FUNCTION_BLOCK FB_Auto_SC
VAR_INPUT
	bEnable				: BOOL;
END_VAR
VAR_OUTPUT
	fPCV				: LREAL;
	fSCV				: LREAL;
	
END_VAR
VAR
	
//Function Blocks
fbPID_payloadpos			: FB_PID_Controller_posref;
fbDeadband_startpos			: FB_Deadband_Auto;
fbDeadband					: FB_Deadband;
fbDisplacementControl_SC	: FB_DisplacementControl_SC;
fbDerivator					: FB_Derivator;

fbClock						: FB_Clock;
fbMUX_selector				: FB_MUX_selector;

//Deadband
fUpperdeadband				: LREAL := 0.5;
fLowerdeadband				: LREAL := 0.14;
fNeutraldeadband			: LREAL := 0.35;
fDeadbandComp_out			: LREAL;

//Outer Loop output
fSC_ClosedLoopSingal		: LREAL;

//VelRef
fWinchVelRefSine			: LREAL;

//Valvesignals
fPCV_set					: LREAL := 1.0;
fPCV_On						: LREAL;
fPCV_Off					: LREAL;

fSCV_startpos				: LREAL;
fSCV_sine					: LREAL;
fSCV_Off					: LREAL;


END_VAR
VAR // added by the converter: edge detectors and wires of the graphical bodies
    _w1 : LREAL;
    _w2 : BOOL;
END_VAR

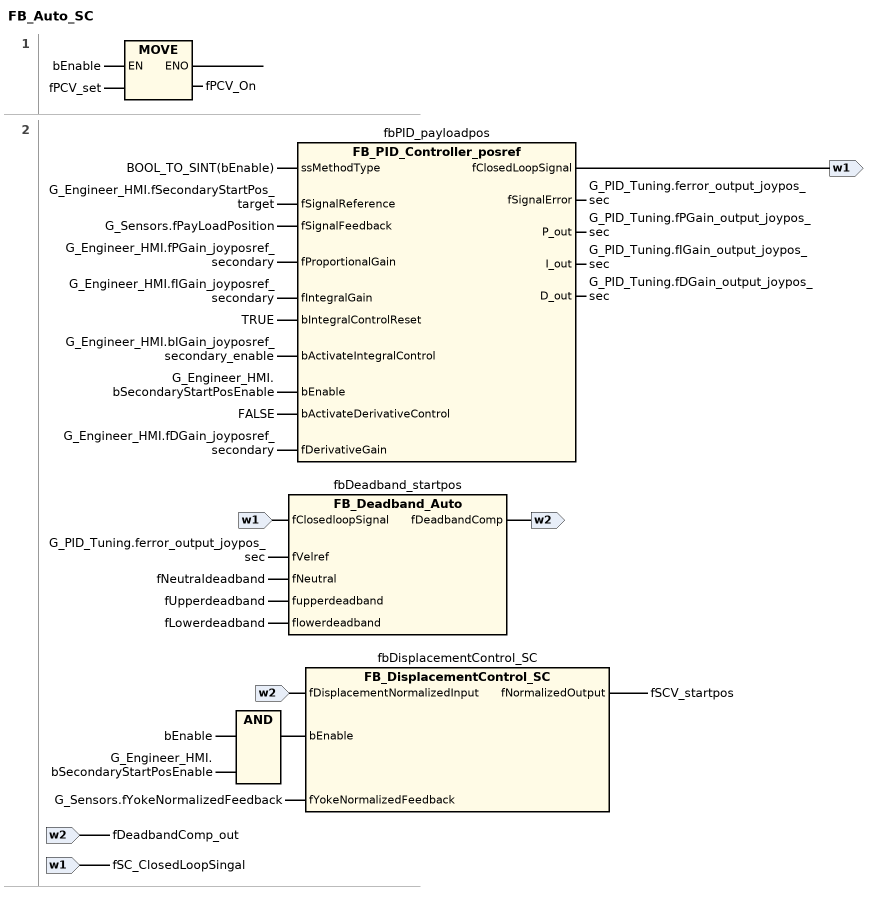
// NETWORK 1
IF bEnable THEN fPCV_On := fPCV_set; END_IF

// NETWORK 2
fbPID_payloadpos(
    ssMethodType := BOOL_TO_SINT(bEnable),
    fSignalReference := G_Engineer_HMI.fSecondaryStartPos_target,
    fSignalFeedback := G_Sensors.fPayLoadPosition,
    fProportionalGain := G_Engineer_HMI.fPGain_joyposref_secondary,
    fIntegralGain := G_Engineer_HMI.fIGain_joyposref_secondary,
    bIntegralControlReset := TRUE,
    bActivateIntegralControl := G_Engineer_HMI.bIGain_joyposref_secondary_enable,
    bEnable := G_Engineer_HMI.bSecondaryStartPosEnable,
    bActivateDerivativeControl := FALSE,
    fDerivativeGain := G_Engineer_HMI.fDGain_joyposref_secondary,
    fSignalError => G_PID_Tuning.ferror_output_joypos_sec,
    P_out => G_PID_Tuning.fPGain_output_joypos_sec,
    I_out => G_PID_Tuning.fIGain_output_joypos_sec,
    D_out => G_PID_Tuning.fDGain_output_joypos_sec); // FB_PID_Controller_posref
fbDeadband_startpos(
    fClosedloopSignal := fbPID_payloadpos.fClosedLoopSignal,
    fVelref := G_PID_Tuning.ferror_output_joypos_sec,
    fNeutral := fNeutraldeadband,
    fupperdeadband := fUpperdeadband,
    flowerdeadband := fLowerdeadband); // FB_Deadband_Auto
fbDisplacementControl_SC(
    fDisplacementNormalizedInput := fbDeadband_startpos.fDeadbandComp,
    bEnable := bEnable AND G_Engineer_HMI.bSecondaryStartPosEnable,
    fYokeNormalizedFeedback := G_Sensors.fYokeNormalizedFeedback); // FB_DisplacementControl_SC
fSCV_startpos := fbDisplacementControl_SC.fNormalizedOutput;
fDeadbandComp_out := fbDeadband_startpos.fDeadbandComp;
fSC_ClosedLoopSingal := fbPID_payloadpos.fClosedLoopSignal;

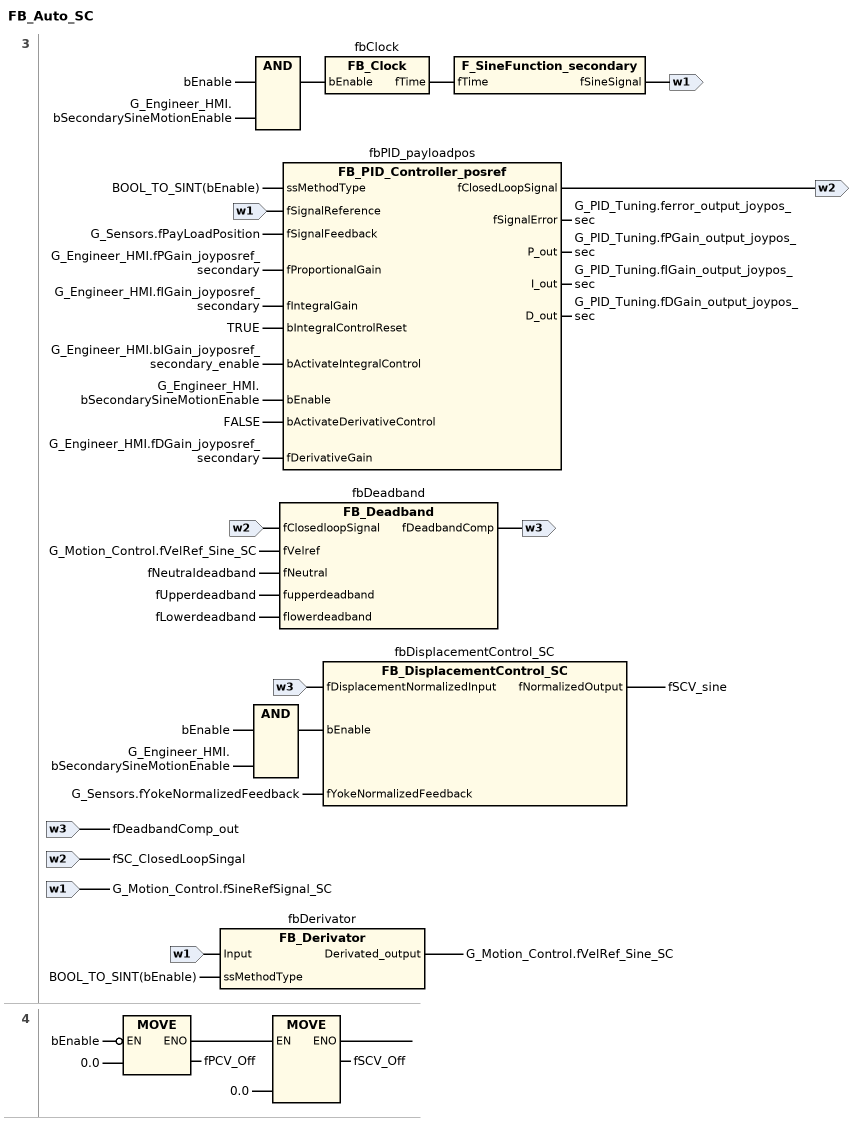
// NETWORK 3
fbClock(bEnable := bEnable AND G_Engineer_HMI.bSecondarySineMotionEnable); // FB_Clock
F_SineFunction_secondary(fTime := fbClock.fTime, fSineSignal => _w1);
fbPID_payloadpos(
    ssMethodType := BOOL_TO_SINT(bEnable),
    fSignalReference := _w1,
    fSignalFeedback := G_Sensors.fPayLoadPosition,
    fProportionalGain := G_Engineer_HMI.fPGain_joyposref_secondary,
    fIntegralGain := G_Engineer_HMI.fIGain_joyposref_secondary,
    bIntegralControlReset := TRUE,
    bActivateIntegralControl := G_Engineer_HMI.bIGain_joyposref_secondary_enable,
    bEnable := G_Engineer_HMI.bSecondarySineMotionEnable,
    bActivateDerivativeControl := FALSE,
    fDerivativeGain := G_Engineer_HMI.fDGain_joyposref_secondary,
    fSignalError => G_PID_Tuning.ferror_output_joypos_sec,
    P_out => G_PID_Tuning.fPGain_output_joypos_sec,
    I_out => G_PID_Tuning.fIGain_output_joypos_sec,
    D_out => G_PID_Tuning.fDGain_output_joypos_sec); // FB_PID_Controller_posref
fbDeadband(
    fClosedloopSignal := fbPID_payloadpos.fClosedLoopSignal,
    fVelref := G_Motion_Control.fVelRef_Sine_SC,
    fNeutral := fNeutraldeadband,
    fupperdeadband := fUpperdeadband,
    flowerdeadband := fLowerdeadband); // FB_Deadband
fbDisplacementControl_SC(
    fDisplacementNormalizedInput := fbDeadband.fDeadbandComp,
    bEnable := bEnable AND G_Engineer_HMI.bSecondarySineMotionEnable,
    fYokeNormalizedFeedback := G_Sensors.fYokeNormalizedFeedback); // FB_DisplacementControl_SC
fSCV_sine := fbDisplacementControl_SC.fNormalizedOutput;
fDeadbandComp_out := fbDeadband.fDeadbandComp;
fSC_ClosedLoopSingal := fbPID_payloadpos.fClosedLoopSignal;
G_Motion_Control.fSineRefSignal_SC := _w1;
fbDerivator(Input := _w1, ssMethodType := BOOL_TO_SINT(bEnable)); // FB_Derivator
G_Motion_Control.fVelRef_Sine_SC := fbDerivator.Derivated_output;

// NETWORK 4
_w2 := NOT bEnable;
IF _w2 THEN fPCV_Off := 0.0; END_IF
IF _w2 THEN fSCV_Off := 0.0; END_IF

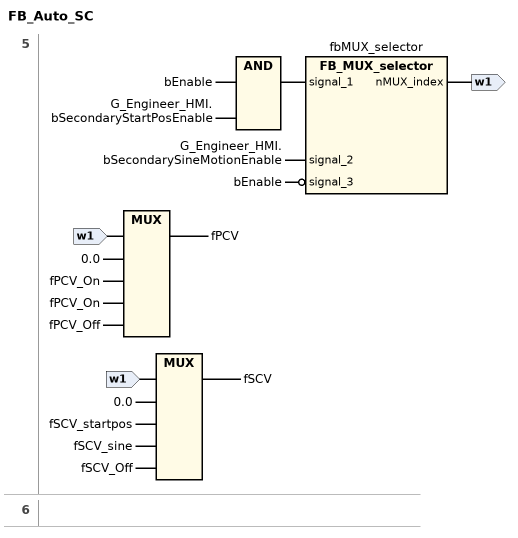
// NETWORK 5
fbMUX_selector(
    signal_1 := bEnable AND G_Engineer_HMI.bSecondaryStartPosEnable,
    signal_2 := G_Engineer_HMI.bSecondarySineMotionEnable,
    signal_3 := NOT bEnable); // FB_MUX_selector
fPCV := MUX(fbMUX_selector.nMUX_index, 0.0, fPCV_On, fPCV_On, fPCV_Off);
fSCV := MUX(fbMUX_selector.nMUX_index, 0.0, fSCV_startpos, fSCV_sine, fSCV_Off);

// NETWORK 6

END_FUNCTION_BLOCK

(* stored: Version 1.1.0.1
   POU FB_Auto_SC: Id {376f8971-d678-4d52-b268-171162ccc33c}, SpecialFunc None *)
